(* IEC 61131-3 sources: SafePLC-Gen-Evaluation/Evaluation Results/P_ID/run_04, 2 files *)

(* ---- io_declarations.st ---- *)
(* ==================================================  *)
(* PLC I/O Variable Declarations — CODESYS 3.5  *)
(* Generated by SafePLC-Gen Multimodal  *)
(* ==================================================  *)

VAR_GLOBAL
    (* --- Analog Inputs ---  *)
    FT_10_Raw                    AT %IW0       : INT := 0;    (* FT-10 — Flow transmitter on upper process line,   *)
    FT_11_Raw                    AT %IW2       : INT := 0;    (* FT-11 — Flow transmitter on lower process line,   *)
    (* --- Analog Outputs ---  *)
    Fv_3_3040_Out                AT %QW0       : INT := 0;    (* Fv-3-3040 — Flow control valve on upper process line  *)
    Fv_3_3041_Out                AT %QW2       : INT := 0;    (* Fv-3-3041 — Flow control valve on lower process line  *)
    (* --- Digital Outputs ---  *)
    XV_ISA_001                   AT %QX0.0     : BOOL := FALSE;    (* XV-ISA-001 — Instrument air supply isolation/regulati  *)
    XV_ISA_002                   AT %QX0.1     : BOOL := FALSE;    (* XV-ISA-002 — Instrument air supply isolation/regulati  *)
END_VAR

(* ---- generated_code.st ---- *)
(* Generated by SafePLC-Gen Multimodal — CODESYS 3.5 *)
(* IEC 61131-3 Structured Text *)
(* Date: 2026-04-25T12:50:22.347857 *)

PROGRAM FlowControl

VAR
    FT_10_Raw                    AT %IW0       : INT := 0;
    FT_11_Raw                    AT %IW2       : INT := 0;
    Fv_3_3040_Out                AT %QW0       : INT := 0;
    Fv_3_3041_Out                AT %QW2       : INT := 0;
    XV_ISA_001                   AT %QX0.0     : BOOL := FALSE;
    XV_ISA_002                   AT %QX0.1     : BOOL := FALSE;
END_VAR

VAR
    FirstScan                    : BOOL := TRUE;

    FT_10_Scaled                 : REAL := 0.0;
    FT_11_Scaled                 : REAL := 0.0;

    FT_10_SP                     : REAL := 50.0;
    FT_11_SP                     : REAL := 50.0;

    FT_10_EU_Min                 : REAL := 0.0;
    FT_10_EU_Span                : REAL := 100.0;
    FT_11_EU_Min                 : REAL := 0.0;
    FT_11_EU_Span                : REAL := 100.0;

    FT_10_HH_SP                  : REAL := 90.0;
    FT_10_H_SP                   : REAL := 80.0;
    FT_10_L_SP                   : REAL := 20.0;
    FT_10_LL_SP                  : REAL := 10.0;
    FT_10_Deadband               : REAL := 2.0;

    FT_11_HH_SP                  : REAL := 90.0;
    FT_11_H_SP                   : REAL := 80.0;
    FT_11_L_SP                   : REAL := 20.0;
    FT_11_LL_SP                  : REAL := 10.0;
    FT_11_Deadband               : REAL := 2.0;

    FT_10_HH                     : BOOL := FALSE;
    FT_10_H                      : BOOL := FALSE;
    FT_10_L                      : BOOL := FALSE;
    FT_10_LL                     : BOOL := FALSE;
    FT_11_HH                     : BOOL := FALSE;
    FT_11_H                      : BOOL := FALSE;
    FT_11_L                      : BOOL := FALSE;
    FT_11_LL                     : BOOL := FALSE;

    (* SR latches initialised with S1=FALSE, R=FALSE so Q1 starts FALSE *)
    FT_10_HH_Latch               : SR := (S1 := FALSE, R := FALSE);
    FT_10_LL_Latch               : SR := (S1 := FALSE, R := FALSE);
    FT_11_HH_Latch               : SR := (S1 := FALSE, R := FALSE);
    FT_11_LL_Latch               : SR := (S1 := FALSE, R := FALSE);

    FT_10_HH_Ack                 : BOOL := FALSE;
    FT_10_LL_Ack                 : BOOL := FALSE;
    FT_11_HH_Ack                 : BOOL := FALSE;
    FT_11_LL_Ack                 : BOOL := FALSE;

    FIC_10_Error                 : REAL := 0.0;
    FIC_10_Integral              : REAL := 0.0;
    FIC_10_Output                : REAL := 0.0;
    FIC_10_Kp                    : REAL := 1.2;
    FIC_10_Ki                    : REAL := 0.05;

    FIC_11_Error                 : REAL := 0.0;
    FIC_11_Integral              : REAL := 0.0;
    FIC_11_Output                : REAL := 0.0;
    FIC_11_Kp                    : REAL := 1.2;
    FIC_11_Ki                    : REAL := 0.05;

    XV_ISA_001_Cmd               : BOOL := FALSE;
    XV_ISA_002_Cmd               : BOOL := FALSE;

    System_Alarm                 : BOOL := FALSE;
END_VAR

IF FirstScan THEN
    Fv_3_3040_Out   := 6554;
    Fv_3_3041_Out   := 6554;
    XV_ISA_001      := FALSE;
    XV_ISA_002      := FALSE;
    FIC_10_Integral := 0.0;
    FIC_11_Integral := 0.0;
    (* Ensure latches start in known de-energised state *)
    FT_10_HH_Latch(S1 := FALSE, R := TRUE);
    FT_10_LL_Latch(S1 := FALSE, R := TRUE);
    FT_11_HH_Latch(S1 := FALSE, R := TRUE);
    FT_11_LL_Latch(S1 := FALSE, R := TRUE);
    FirstScan       := FALSE;
    RETURN;
END_IF;

FT_10_Scaled := ((INT_TO_REAL(FT_10_Raw) - 6554.0) / (32767.0 - 6554.0)) * FT_10_EU_Span + FT_10_EU_Min;
FT_11_Scaled := ((INT_TO_REAL(FT_11_Raw) - 6554.0) / (32767.0 - 6554.0)) * FT_11_EU_Span + FT_11_EU_Min;

IF FT_10_Scaled >= FT_10_HH_SP THEN
    FT_10_HH := TRUE;
ELSIF FT_10_Scaled <= (FT_10_HH_SP - FT_10_Deadband) THEN
    FT_10_HH := FALSE;
END_IF;

IF FT_10_Scaled >= FT_10_H_SP THEN
    FT_10_H := TRUE;
ELSIF FT_10_Scaled <= (FT_10_H_SP - FT_10_Deadband) THEN
    FT_10_H := FALSE;
END_IF;

IF FT_10_Scaled <= FT_10_L_SP THEN
    FT_10_L := TRUE;
ELSIF FT_10_Scaled >= (FT_10_L_SP + FT_10_Deadband) THEN
    FT_10_L := FALSE;
END_IF;

IF FT_10_Scaled <= FT_10_LL_SP THEN
    FT_10_LL := TRUE;
ELSIF FT_10_Scaled >= (FT_10_LL_SP + FT_10_Deadband) THEN
    FT_10_LL := FALSE;
END_IF;

FT_10_HH_Latch(S1 := FT_10_HH,
               R  := (FT_10_HH_Ack AND NOT FT_10_HH));

FT_10_LL_Latch(S1 := FT_10_LL,
               R  := (FT_10_LL_Ack AND NOT FT_10_LL));

IF FT_11_Scaled >= FT_11_HH_SP THEN
    FT_11_HH := TRUE;
ELSIF FT_11_Scaled <= (FT_11_HH_SP - FT_11_Deadband) THEN
    FT_11_HH := FALSE;
END_IF;

IF FT_11_Scaled >= FT_11_H_SP THEN
    FT_11_H := TRUE;
ELSIF FT_11_Scaled <= (FT_11_H_SP - FT_11_Deadband) THEN
    FT_11_H := FALSE;
END_IF;

IF FT_11_Scaled <= FT_11_L_SP THEN
    FT_11_L := TRUE;
ELSIF FT_11_Scaled >= (FT_11_L_SP + FT_11_Deadband) THEN
    FT_11_L := FALSE;
END_IF;

IF FT_11_Scaled <= FT_11_LL_SP THEN
    FT_11_LL := TRUE;
ELSIF FT_11_Scaled >= (FT_11_LL_SP + FT_11_Deadband) THEN
    FT_11_LL := FALSE;
END_IF;

FT_11_HH_Latch(S1 := FT_11_HH,
               R  := (FT_11_HH_Ack AND NOT FT_11_HH));

FT_11_LL_Latch(S1 := FT_11_LL,
               R  := (FT_11_LL_Ack AND NOT FT_11_LL));

FIC_10_Error    := FT_10_SP - FT_10_Scaled;
FIC_10_Integral := FIC_10_Integral + (FIC_10_Ki * FIC_10_Error);
IF FIC_10_Integral > 100.0 THEN
    FIC_10_Integral := 100.0;
ELSIF FIC_10_Integral < 0.0 THEN
    FIC_10_Integral := 0.0;
END_IF;
FIC_10_Output := (FIC_10_Kp * FIC_10_Error) + FIC_10_Integral;
IF FIC_10_Output > 100.0 THEN
    FIC_10_Output := 100.0;
ELSIF FIC_10_Output < 0.0 THEN
    FIC_10_Output := 0.0;
END_IF;
Fv_3_3040_Out := REAL_TO_INT(6554.0 + (FIC_10_Output / 100.0) * (32767.0 - 6554.0));

FIC_11_Error    := FT_11_SP - FT_11_Scaled;
FIC_11_Integral := FIC_11_Integral + (FIC_11_Ki * FIC_11_Error);
IF FIC_11_Integral > 100.0 THEN
    FIC_11_Integral := 100.0;
ELSIF FIC_11_Integral < 0.0 THEN
    FIC_11_Integral := 0.0;
END_IF;
FIC_11_Output := (FIC_11_Kp * FIC_11_Error) + FIC_11_Integral;
IF FIC_11_Output > 100.0 THEN
    FIC_11_Output := 100.0;
ELSIF FIC_11_Output < 0.0 THEN
    FIC_11_Output := 0.0;
END_IF;
Fv_3_3041_Out := REAL_TO_INT(6554.0 + (FIC_11_Output / 100.0) * (32767.0 - 6554.0));

(* Instrument air isolation valves — open when no HH or LL alarm latched *)
XV_ISA_001_Cmd := NOT (FT_10_HH_Latch.Q1 OR FT_10_LL_Latch.Q1 OR FT_11_HH_Latch.Q1 OR FT_11_LL_Latch.Q1);
XV_ISA_002_Cmd := XV_ISA_001_Cmd;
XV_ISA_001     := XV_ISA_001_Cmd;
XV_ISA_002     := XV_ISA_002_Cmd;

System_Alarm :=
    FT_10_HH_Latch.Q1 OR FT_10_LL_Latch.Q1 OR
    FT_10_H            OR FT_10_L            OR
    FT_11_HH_Latch.Q1 OR FT_11_LL_Latch.Q1 OR
    FT_11_H            OR FT_11_L;

END_PROGRAM
